Staubli VAL3: GetSerialNumber.pgx

program GetSerialNumber(string& answer)
begin
  //*******************************************************************************
  //*   ______
  //*  / _____) /|
  //* | |      / /
  //* | | /\  / /
  //* | | \ \/ /  _      Copyright (c) KEOLABS, 2016
  //* | |  \__/  | |        http://www.keolabs.com
  //* | |________| |
  //*  \__________/
  //*
  //********************************************************************************
  //*@file          : GetSerialNumber
  //*@author        : Yves Ragot
  //*@version       : $Id: GetSerialNumber.pgx 1198 2016-10-07 06:48:14Z yves $
  //*@brief         : Get Serial Number of the arm
  //*
  //*******************************************************************************/

  answer = left(getVersion("ArmSN"), 20)

end
